TYPE ST_ItemPK2_OUT1 :
STRUCT
	Identity		:ST_Identity_PK2_OUT1;
	ItemState		:STRING;
	RejectReason	:ST_RejectReason_PK2_OUT1;
	logs			:ST_logs_PK2_OUT1;
	NoRead			:STRING;
END_STRUCT
END_TYPE

(* stored: Version 1.1.0.1, ProductVersion 3.1.4024.13
   DUT ST_ItemPK2_OUT1: Id {fe2387d3-36f1-4b28-9c2e-232560710f5a} *)
